# EPICS autosave request: iocBoot/iocNSLS2_IC/auto_settings.req
file "NSLS2_EM_settings.req",          P=$(P), R=$(R)
file "quadEM_IOC_settings.req",        P=$(P), R=$(R)
